PROGRAM MAIN
VAR
	//FBs
	fbPlant: FB_Plant;
	Ctrl_data_plant : Plant_CTRL;
	
	fbConveyorEntry : FB_Conveyor;
	
	fbSorter : FB_Sorter;
	
	// Control modules call
	cmVision : CM_VisionSensor;
	Ctrl_data_vision : CM_Vision_UDT;
	
	cmConveyor1 : CM_DO;
	cmConveyor2 : CM_DO;
	Ctrl_data_Conveyor1 : CM_DO_UDT;
	Ctrl_data_Conveyor2 : CM_DO_UDT;
	
	cmAtExit : CM_DIN;
	Ctrl_data_exit : CM_DIN_UDT;
	
	cmSorter1 : CM_DO;
	Crtl_data_sorter1 : CM_DO_UDT;
	cmSorter2 : CM_DO;
	Crtl_data_sorter2 : CM_DO_UDT;
	cmSorter3 : CM_DO;
	Crtl_data_sorter3 : CM_DO_UDT;
	
	cmStopBlade : CM_DO;
	crtl_data_StopBlade : CM_DO_UDT;
	
	cmEmitter : CM_DO;
	ctrl_data_emitter : CM_DO_UDT;
	
END_VAR

VAR_IN_OUT
	
END_VAR


fbPlant(
	bAuto_IN:= FIO.bAuto, 
	bManual_IN:= FIO.bManual,
	bStart_IN := FIO.bStart,
	bStop_IN := FIO.bStop,
	bReset_IN := FIO.bReset,
	bEmgStop_IN := FIO.bEmgStop,
 
	bAuto_OUT=> , 
	bManual_OUT=> ,
 
	PlantCtrl:= Ctrl_data_plant);
	
IF fbPlant.bEmgStop_IN THEN
	fbConveyorEntry(
		control_data := Ctrl_data_plant,
		control_data_vision := Ctrl_data_vision,
		control_data_Conveyor1 := Ctrl_data_Conveyor1,
		control_data_StopBlade := crtl_data_StopBlade,
		control_data_emitter := ctrl_data_emitter
		);	
	
	fbSorter(
		control_data := Ctrl_data_plant,
		control_data_vision := Ctrl_data_vision,
		control_data_Conveyor2 := Ctrl_data_Conveyor2,
		control_data_sorter1 := Crtl_data_sorter1,
		control_data_sorter2 := Crtl_data_sorter2,
		control_data_sorter3 := Crtl_data_sorter3,
		control_data_atExit := Ctrl_data_exit,
	
	);	
END_IF	



//// CM Calls
cmConveyor1( 
	Control_data_DO := Ctrl_data_Conveyor1,
	
   	PO_HighCommand => FIO.bConveyorEntry_out
	); 
 
cmConveyor2(
	Control_data_DO := Ctrl_data_Conveyor2,
	PO_HighCommand => FIO.bConveyorExit_out
	);
	
cmAtExit(
	PI_autoHigh := FIO.bAtExit,
	Control_data := Ctrl_data_exit);

	
cmVision(
	SensorInput := FIO.iVisionSensor,
	control_data_vision := Ctrl_data_Vision);
	
cmSorter1(
	Control_data_DO := Crtl_data_sorter1,
	PO_HighCommand => FIO.bSorter_1_out, 
	PO_HighCommand => FIO.bSorter_1_turn
	);
cmSorter2(
	Control_data_DO := Crtl_data_sorter2,
	PO_HighCommand => FIO.bSorter_2_out, 
	PO_HighCommand => FIO.bSorter_2_turn
	);
	
cmSorter3(
	Control_data_DO := Crtl_data_sorter3,
	PO_HighCommand => FIO.bSorter_3_out,
	PO_HighCommand => FIO.bSorter_3_turn
	);
	
cmStopBlade(
	Control_data_DO := crtl_data_StopBlade,
	PO_HighCommand => FIO.bStopBlade
	);
cmEmitter(
	PO_HighCommand => FIO.bEmitter,
	Control_data_DO := ctrl_data_emitter
	);

END_PROGRAM

(* stored: Version 1.1.0.1, ProductVersion 3.1.4024.13
   POU MAIN: Id {54fc3697-1197-40f3-acf2-4a0b47230f51}, SpecialFunc None *)
